FUNCTION FC_4strConcatSeparator : T_DEFAULT_STR		// Concatenates 4 strings with given separator
VAR_INPUT
	iSeparator:		STRING := IING.STRING_UNDERSCORE;
	iStr1:			T_DEFAULT_STR;
	iStr2:			T_DEFAULT_STR;
	iStr3:			T_DEFAULT_STR;
	iStr4:			T_DEFAULT_STR;
END_VAR

FC_4strConcatSeparator := FC_2strConcatSeparator(iSeparator := iSeparator,
	iStr1 := FC_3strConcatSeparator(iSeparator := iSeparator, iStr1 := iStr1, iStr2 := iStr2, iStr3 := iStr3), iStr2 := iStr4);

END_FUNCTION

(* stored: Version 1.1.0.1, ProductVersion 3.1.4026.18
   POU FC_4strConcatSeparator: Id {c994d032-4809-4f26-9023-944e4d570efe}, SpecialFunc None *)
